// TIA Portal V21 export
DATA_BLOCK "Motore"   // DB11
{ S7_Optimized_Access := 'TRUE' }
// stored: MemoryReserve 100
   VAR RETAIN
      "M" : Array[0.."K_NumMotore"] of "Std_stMotore";
   END_VAR
   VAR
      Funzioni : Struct
         DefaultPrm : Bool := FALSE;   // Ripristino dei dati iniziali
         TuttiInAutoMode : Bool := FALSE;
      END_STRUCT;
   END_VAR
BEGIN
   // "M"[0] : NON USARE
   "M"[0].HMI.STW1 := 16#0000;
   "M"[0].HMI.CTW1 := 16#0000;
END_DATA_BLOCK
